PROGRAM HMI_WEB_dataConver
VAR
END_VAR

Hmi_Web.Car_pos := Axis.FeedCar.Pos;

END_PROGRAM

(* stored: Version 1.1.0.1, ProductVersion 3.1.4026.13
   POU HMI_WEB_dataConver: Id {173a9c07-f878-4e60-89ac-7c28f0373126}, SpecialFunc None *)
